{attribute addProperty BoxType "EL6688-0000-0022"}
{attribute addProperty Id "External_SyncAT %I*External_Sync_07348351192240WcStateAT %I*WcState_F855686C1620InfoDataAT %I*InfoData_0BDED7BF144180"}
{attribute addProperty CRC "866557102"}
{attribute addProperty SizeInBites "352"}
{attribute addProperty SizeInBytes "44"}
TYPE EL6688_7BDEAC92 :
STRUCT
	{attribute addProperty Name "External_Sync"}
	External_Sync : External_Sync_07348351;
	{attribute addProperty Name "WcState"}
	WcState : WcState_F855686C;
	{attribute addProperty Name "InfoData"}
	InfoData : InfoData_0BDED7BF;
END_STRUCT
END_TYPE

(* stored: Version 1.2.0.0, ProductVersion 3.1.4024.9
   DUT EL6688_7BDEAC92: Id {9e3646fa-905d-45c1-a322-7f5228a003ea} *)
